SUBAPPLICATION Uebung_006f_RS_AX (* Exercise for FB_RS_T_FF (Reset-Dominant Toggle Flip-Flop) *)
  (* Standard: 61499-2; Description: Copyright (c) 2026 Meisterschulen am Ostbahnhof *)
  (* Version 1.0, 2026-05-07, Gemini CLI, Meisterschulen am Ostbahnhof *)
  PACKAGE Uebungen;
  IMPORT logiBUS::io::DI::logiBUS_DI::Input_I1;
  IMPORT logiBUS::io::DI::logiBUS_DI::Input_I2;
  IMPORT logiBUS::io::DI::logiBUS_DI::Input_I3;
  IMPORT logiBUS::io::DQ::logiBUS_DO::Output_Q1;
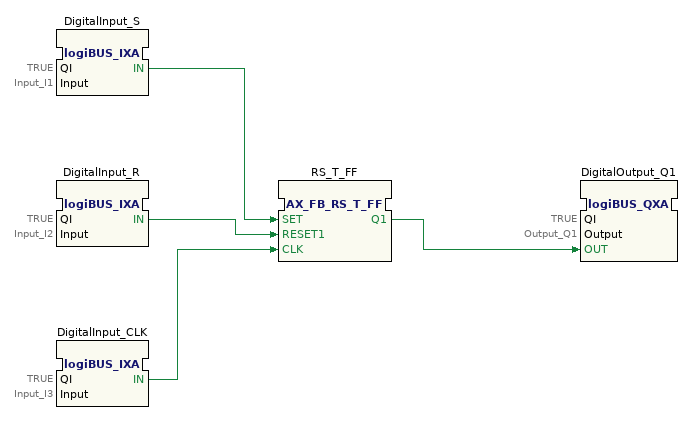
  FBS
    DigitalInput_S : logiBUS::io::DI::logiBUS_IXA(QI := TRUE, Input := Input_I1);
    DigitalInput_R : logiBUS::io::DI::logiBUS_IXA(QI := TRUE, Input := Input_I2);
    DigitalInput_CLK : logiBUS::io::DI::logiBUS_IXA(QI := TRUE, Input := Input_I3);
    RS_T_FF : adapter::bistableElements::AX_FB_RS_T_FF;
    DigitalOutput_Q1 : logiBUS::io::DQ::logiBUS_QXA(QI := TRUE, Output := Output_Q1);
  END_FBS
  ADAPTER_CONNECTIONS
    DigitalInput_S.IN TO RS_T_FF.SET;
    DigitalInput_R.IN TO RS_T_FF.RESET1;
    DigitalInput_CLK.IN TO RS_T_FF.CLK;
    RS_T_FF.Q1 TO DigitalOutput_Q1.OUT;
  END_CONNECTIONS
END_SUBAPPLICATION
